(* Logix 5000 project; controller ChiaDynamix Emulate 5570 rev 30.12; software revision 30.00 *)

TASK T00_MainTask (continuous, watchdog 500 ms) : P00_MainProgram

MODULES
   Local : Emulate 5570 (ICP 2, rev 30.12)
      Entradas_Digitales : 1756-IB16 (ICP 3, rev 3.1, Input RPI 20 ms)
      Salidas_Digitales : vendor 1 type 7 code 16 (ICP 4, rev 3.1, Output RPI 20 ms)
      PLC2 : Emulate 5570 (ICP 5, rev 30.1, $76991c4e$ RPI 20 ms, $e229f641$ RPI 20 ms, $a5fb9b3a$ RPI 20 ms, $28fe76d7$ RPI 20 ms, $af09fea8$ RPI 20 ms, $a0c3347f$ RPI 20 ms, $42741be5$ RPI 20 ms, $de8c326e$ RPI 20 ms, $741f7ed2$ RPI 20 ms)
      PLC_Seguridad : Emulate 5570 (ICP 6, rev 30.1, $262d7f5a$ RPI 20 ms)
END_MODULES

VAR_GLOBAL   (* controller tags *)
   CIL_PREN_001 : ALIAS FOR Local:4:I.Data.1;   // Cilindro de Prensa Hidráulica
   Controles_Permisivos_Consumidos : DINT;   // Señal de seguridad que se recibe del PLC de Seguridad e indica que algún elemento de seguridad ha sido activado
   Count_Baldosas_Consumido : DINT;   // Memoria Virtual del Contador de baldosas que se recibe del PLC2
   Count_Cajas_Consumido : DINT;   // Memoria Virtual del Contador de cajas que se recibe del PLC2
   FAB_CER_AUTO_001 : DINT; {produced}   // Botón de Automático PLC1
   FAB_CER_CORTINAS_SEGURIDAD_Producido : DINT := 1; {produced}   // Cortina de Seguridad PLC1
   FAB_CER_EME_001 : DINT := 1; {produced}   // Botón de Emergencia PLC1
   FAB_CER_RES_001 : DINT; {produced}   // Botón de Reset PLC1
   FAB_CER_STP_001 : DINT; {produced}   // Botón de Parada PLC1
   FAB_CER_STR_001 : DINT; {produced}   // Botón de Arranque PLC1
   FAB_CER_TAPETE_SEGURIDAD_Producido : DINT := 1; {produced}   // Tapete de Seguridad PLC1
   MA_ESMAL_001 : ALIAS FOR Local:4:I.Data.2;   // Máquina de Esmaltado
   MA_HORNO_001 : ALIAS FOR Local:4:I.Data.4;   // Señal de Secado (Indica que Horno ya acabó)
   MA_IMPR_001 : ALIAS FOR Local:4:I.Data.3;   // Máquina de Impresión de Patrones
   MOT_BAND_001 : ALIAS FOR Local:4:I.Data.0;   // Motor Banda transportadora
   POS_BAN_IMP : ALIAS FOR Local:3:I.Data.14;   // Sensor de posición ubicado en banda de proceso de impresión
   POS_BAN_PREN : ALIAS FOR Local:3:I.Data.12;   // Sensor de posición ubicado en banda de prensa
   POS_BAND_ESMAL : ALIAS FOR Local:3:I.Data.13;   // Sensor de posición ubicado en banda de proceso de esmaltado
   POS_BAND_HORNO1 : ALIAS FOR Local:3:I.Data.15;   // Sensor de posición ubicado en banda al inicio del proceso del Horno
   POS_BAND_HORNO2 : ALIAS FOR Local:3:I.Data.16;   // Sensor de posición ubicado en banda a la salida del proceso del Horno
   PREN_ABAJO : ALIAS FOR Local:3:I.Data.9;   // Sensor de posición ubicado en prensa abajo
   PREN_ARRIBA : ALIAS FOR Local:3:I.Data.7;   // Sensor de posición ubicado en prensa arrriba
   Q : BOOL[32] := ([10] := 1);
        [2]   // Memoria virtual que activa el cilindro de prensa (A+)
        [4]   // Memoria Virtual que activa Motor
        [7]   // Memoria Virtual que activa Motor
        [3]   // Memoria virtual que desactiva el cilindro de prensa (A-)
        [5]   // Memoria Virtual que activa Motor y Máquina de Esmaltado
        [6]   // Memoria virtual que activa Máquina de Impresión de Patrones
        [8]   // Memoria Virtual que activa Horno
   Q10_Consumido : DINT;   // Memoria Virtual Consumida que se recibe desde el PLC2
   Q13_Consumido : DINT;   // Memoria Virtual Q13 que se recibe del PLC2
   Q16_Consumido : DINT;   // Memoria Virtual Q16 que se recibe del PLC2
   Q17_Consumido : DINT;   // Memoria Virtual Q17 que se recibe del PLC2
   Q1_Producido : DINT; {produced}   // Memoria Virtual que activa Motor
   Q9_Producido : DINT; {produced}   // Memoria Virtual que activa Motor
   SEN_PESO : ALIAS FOR Local:3:I.Data.8;   // Sensor de peso encargado de medir materia prima
   SEN_PRESION : ALIAS FOR Local:3:I.Data.10;   // Sensor de Presión de la prensa
   SEN_TEMP : ALIAS FOR Local:3:I.Data.11;   // Sensor de tempartura del Horno
   SIGNAL_APILADO1_Consumido : DINT;   // Señal recibida del PLC2 que indica que la rutina de apilamiento de baldosas ha finalizado
   SIGNAL_ECOPLAT_Consumido : DINT;   // Señal que se recibe del PLC2 e indica si el proceso de Envoltura ya finalizó
   SIGNAL_HORNO : BOOL;   // Señal que indica que el proceso de secado finalizó
   SIGNAL_IMP : BOOL;   // Señal que indica que ya finalizó proceso de impresión
   SIGNAL_MAINT_Producido : DINT; {produced}   // Señal que indica que se está realizando una operación de mantenimiento
   SIGNAL_ROUT2_Consumido : DINT;   // Señal recibida del PLC2 que indica que la rutina del robot2 ha finalizado
   SIGNAL_STP : BOOL;   // Señal que indica que el Botón de Stop ha sido presionado
   TIMER : TIMER[6] := ([0].PRE := 30000, [1].PRE := 30000);
        [0]   // Timer de Proceso de Impresión
        [1]   // Timer de Proceso de Secado (Horno)
END_VAR

PROGRAM P00_MainProgram   (* main routine R00_MainRoutine *)
VAR
   SIGNAL_EMERGENCY : BOOL;   // El botón de Emergencia está activo
END_VAR

ROUTINE R00_MainRoutine   (* ladder *)
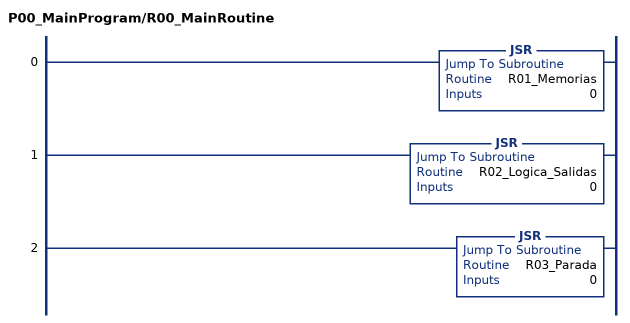
   0: JSR(R01_Memorias,0);
   1: JSR(R02_Logica_Salidas,0);
   2: JSR(R03_Parada,0);
END_ROUTINE

ROUTINE R01_Memorias   (* ladder *)
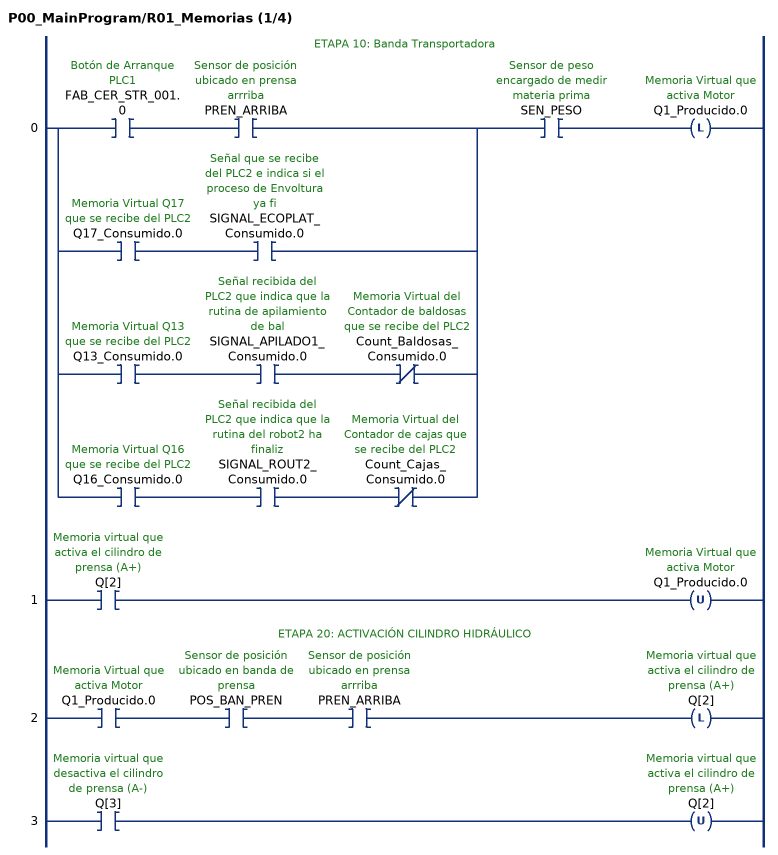
   // ETAPA 10: Banda Transportadora
   0: [XIC(FAB_CER_STR_001.0) XIC(PREN_ARRIBA) ,XIC(Q17_Consumido.0) XIC(SIGNAL_ECOPLAT_Consumido.0) ,XIC(Q13_Consumido.0) XIC(SIGNAL_APILADO1_Consumido.0) XIO(Count_Baldosas_Consumido.0) ,XIC(Q16_Consumido.0) XIC(SIGNAL_ROUT2_Consumido.0) XIO(Count_Cajas_Consumido.0) ]XIC(SEN_PESO)OTL(Q1_Producido.0);
   1: XIC(Q[2])OTU(Q1_Producido.0);
   // ETAPA 20: ACTIVACIÓN CILINDRO HIDRÁULICO
   2: XIC(Q1_Producido.0)XIC(POS_BAN_PREN)XIC(PREN_ARRIBA)OTL(Q[2]);
   3: XIC(Q[3])OTU(Q[2]);
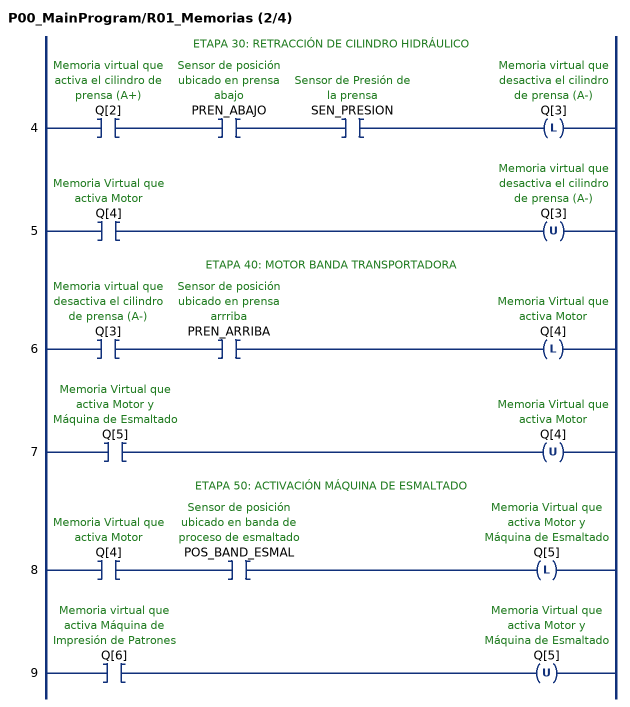
   // ETAPA 30: RETRACCIÓN DE CILINDRO HIDRÁULICO
   4: XIC(Q[2])XIC(PREN_ABAJO)XIC(SEN_PRESION)OTL(Q[3]);
   5: XIC(Q[4])OTU(Q[3]);
   // ETAPA 40: MOTOR BANDA TRANSPORTADORA
   6: XIC(Q[3])XIC(PREN_ARRIBA)OTL(Q[4]);
   7: XIC(Q[5])OTU(Q[4]);
   // ETAPA 50: ACTIVACIÓN MÁQUINA DE ESMALTADO
   8: XIC(Q[4])XIC(POS_BAND_ESMAL)OTL(Q[5]);
   9: XIC(Q[6])OTU(Q[5]);
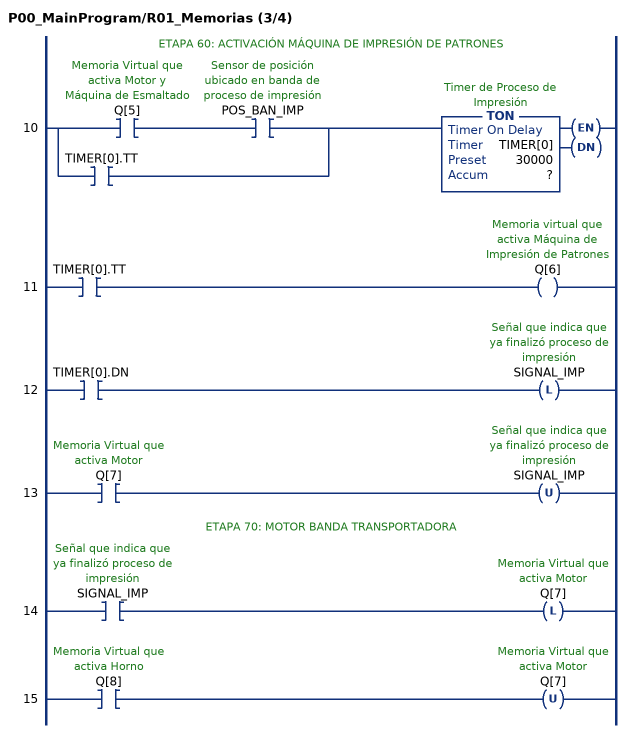
   // ETAPA 60: ACTIVACIÓN MÁQUINA DE IMPRESIÓN DE PATRONES
   10: [XIC(Q[5]) XIC(POS_BAN_IMP) ,XIC(TIMER[0].TT) ]TON(TIMER[0],?,?);
   11: XIC(TIMER[0].TT)OTE(Q[6]);
   12: XIC(TIMER[0].DN)OTL(SIGNAL_IMP);
   13: XIC(Q[7])OTU(SIGNAL_IMP);
   // ETAPA 70: MOTOR BANDA TRANSPORTADORA
   14: XIC(SIGNAL_IMP)OTL(Q[7]);
   15: XIC(Q[8])OTU(Q[7]);
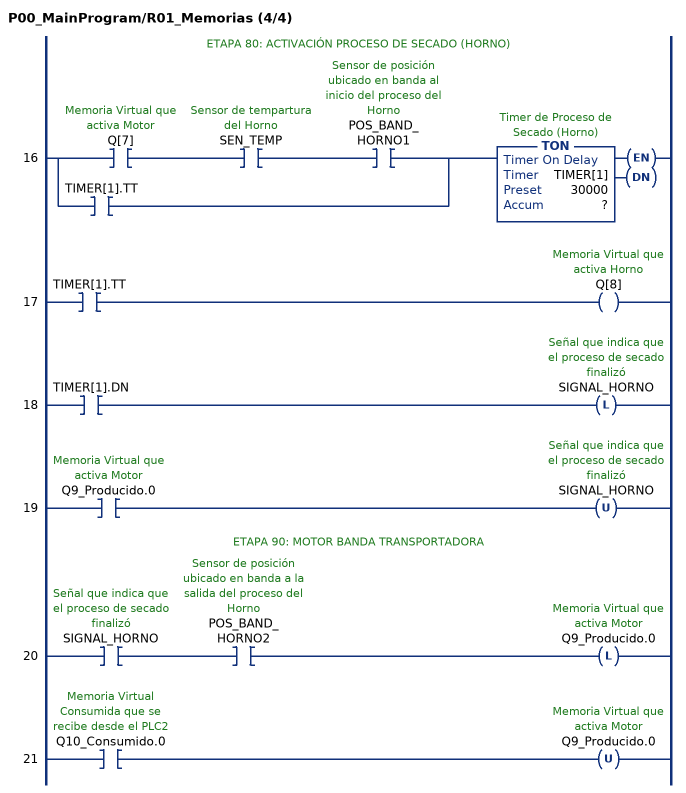
   // ETAPA 80: ACTIVACIÓN PROCESO DE SECADO (HORNO)
   16: [XIC(Q[7]) XIC(SEN_TEMP) XIC(POS_BAND_HORNO1) ,XIC(TIMER[1].TT) ]TON(TIMER[1],?,?);
   17: XIC(TIMER[1].TT)OTE(Q[8]);
   18: XIC(TIMER[1].DN)OTL(SIGNAL_HORNO);
   19: XIC(Q9_Producido.0)OTU(SIGNAL_HORNO);
   // ETAPA 90: MOTOR BANDA TRANSPORTADORA
   20: XIC(SIGNAL_HORNO)XIC(POS_BAND_HORNO2)OTL(Q9_Producido.0);
   21: XIC(Q10_Consumido.0)OTU(Q9_Producido.0);
END_ROUTINE

ROUTINE R02_Logica_Salidas   (* ladder *)
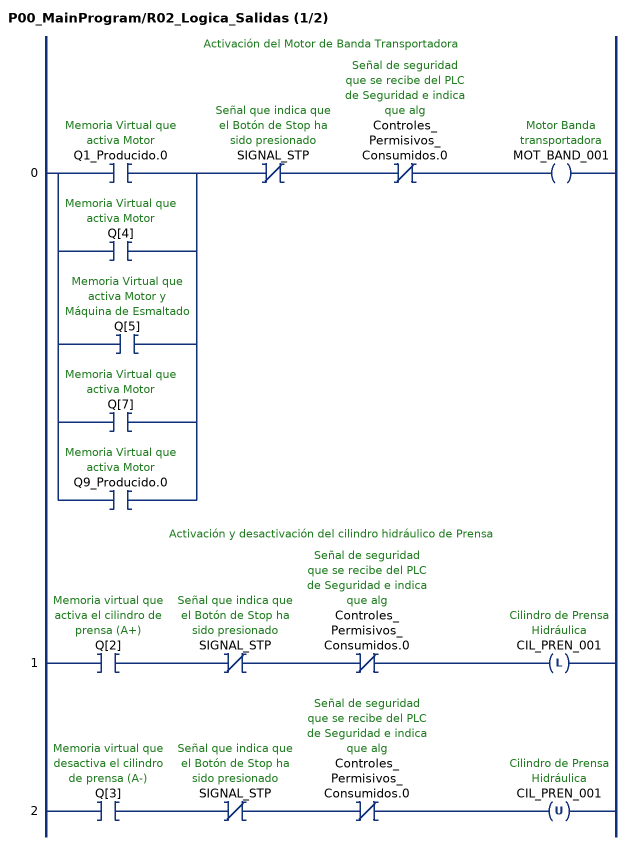
   // Activación del Motor de Banda Transportadora
   0: [XIC(Q1_Producido.0) ,XIC(Q[4]) ,XIC(Q[5]) ,XIC(Q[7]) ,XIC(Q9_Producido.0) ]XIO(SIGNAL_STP)XIO(Controles_Permisivos_Consumidos.0)OTE(MOT_BAND_001);
   // Activación y desactivación del cilindro hidráulico de Prensa
   1: XIC(Q[2])XIO(SIGNAL_STP)XIO(Controles_Permisivos_Consumidos.0)OTL(CIL_PREN_001);
   2: XIC(Q[3])XIO(SIGNAL_STP)XIO(Controles_Permisivos_Consumidos.0)OTU(CIL_PREN_001);
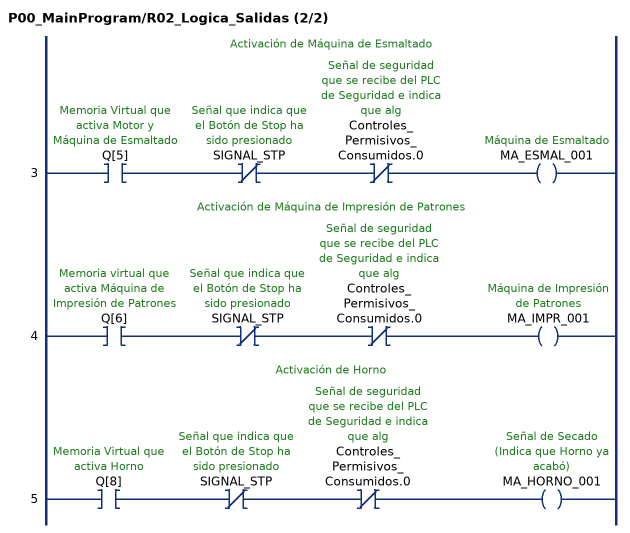
   // Activación de Máquina de Esmaltado
   3: XIC(Q[5])XIO(SIGNAL_STP)XIO(Controles_Permisivos_Consumidos.0)OTE(MA_ESMAL_001);
   // Activación de Máquina de Impresión de Patrones
   4: XIC(Q[6])XIO(SIGNAL_STP)XIO(Controles_Permisivos_Consumidos.0)OTE(MA_IMPR_001);
   // Activación de Horno
   5: XIC(Q[8])XIO(SIGNAL_STP)XIO(Controles_Permisivos_Consumidos.0)OTE(MA_HORNO_001);
END_ROUTINE

ROUTINE R03_Parada   (* ladder *)
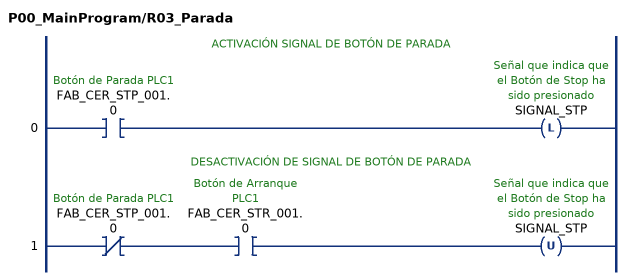
   // ACTIVACIÓN SIGNAL DE BOTÓN DE PARADA
   0: XIC(FAB_CER_STP_001.0)OTL(SIGNAL_STP);
   // DESACTIVACIÓN DE SIGNAL DE BOTÓN DE PARADA
   1: XIO(FAB_CER_STP_001.0)XIC(FAB_CER_STR_001.0)OTU(SIGNAL_STP);
END_ROUTINE
END_PROGRAM
